FUNCTION Convert_BOOL_TO_LREAL : BOOL
VAR_INPUT
	in : BOOL;
	out : REFERENCE TO LREAL;
END_VAR

out := BOOL_TO_LREAL(in);
Convert_BOOL_TO_LREAL := TRUE;

END_FUNCTION

(* stored: Version 1.1.0.1, ProductVersion 3.1.4024.12
   POU Convert_BOOL_TO_LREAL: Id {adb89cf5-c2b2-42dd-8ede-d86a0a994a5b}, SpecialFunc None *)
